INTERFACE I_ALARM_HANDLER

METHOD RegisterAlarm : REFERENCE TO FBA_ALARM_HANDLER
VAR_INPUT
	Alarm : REFERENCE TO FB_ALARM;
	Prefix : STRING := '';
	Update : BOOL := TRUE;
END_VAR
END_METHOD

END_INTERFACE

(* stored: Version 1.1.0.1, ProductVersion 3.1.4024.12
   Itf I_ALARM_HANDLER: Id {5c994d0e-8085-4560-9226-945aa16ffed2}
   Method RegisterAlarm: Id {3356dcaa-b4e3-4ea5-ac44-9fb7255bfd66} *)
